FUNCTION_BLOCK FB_AvanzarAlimentador_SFC

VAR_IN_OUT
	   TpoAlimentador: TIME;
	   FaltaMaterial: BOOL;
END_VAR

VAR_INPUT
    // SFC-Flags
    SFCPause: BOOL;
    SFCReset: BOOL;
    
    // Indicadores de sincronizacion
    Ack: BOOL := TRUE;
    Execute: BOOL;
 
    // Entradas
    AlimentadorDelante: BOOL;
	PulsadorMarcha: BOOL; 
END_VAR
VAR_OUTPUT
    // Indicadores de sincronizacion
    Done: BOOL;
    Ready: BOOL;
	Fallo: BOOL;
    // Salidas
   AlimentadorAvanza: BOOL;
END_VAR
VAR
END_VAR

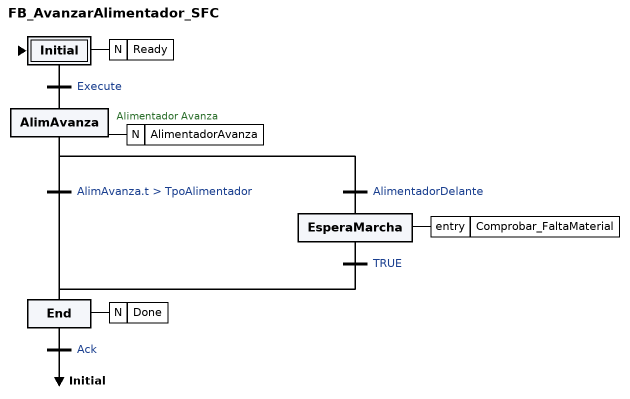
INITIAL_STEP Initial:
    Ready(N);
END_STEP
TRANSITION FROM Initial TO AlimAvanza
    := Execute;
END_TRANSITION
// Alimentador Avanza
STEP AlimAvanza:
    AlimentadorAvanza(N);
END_STEP
TRANSITION FROM AlimAvanza TO End
    := AlimAvanza.t > TpoAlimentador;
END_TRANSITION
TRANSITION FROM AlimAvanza TO EsperaMarcha
    := AlimentadorDelante;
END_TRANSITION
STEP EsperaMarcha:
    Comprobar_FaltaMaterial(P1);  // entry action
END_STEP
TRANSITION FROM EsperaMarcha TO End
    := TRUE;
END_TRANSITION
STEP End:
    Done(N);
END_STEP
TRANSITION FROM End TO Initial
    := Ack;
END_TRANSITION

ACTION Comprobar_FaltaMaterial:
FaltaMaterial := TRUE;
END_ACTION

END_FUNCTION_BLOCK

(* stored: Version 1.1.0.1, ProductVersion 3.1.4024.12
   POU FB_AvanzarAlimentador_SFC: Id {7127f594-2a12-4c1f-91b0-cf4f6d8e670a}, SpecialFunc None
   Action Comprobar_FaltaMaterial: Id {068257fb-c5b6-431c-aade-5b58709e110f} *)
